INTERFACE I_HE_SolidAttenuatorAttentuationLengthDatabase EXTENDS I_Fallible


METHOD GetAttenuationLength
VAR_INPUT
    PhotonEnergy : I_QuantityLREAL;
    MaterialName : T_MaxString;
    AttenuationLengthOutput : I_QuantityLREALPublic;
END_VAR
END_METHOD

END_INTERFACE

(* stored: Version 1.1.0.1
   Itf I_HE_SolidAttenuatorAttentuationLengthDatabase: Id {06dfad59-b310-4aa0-bb9c-06b6bb0d52ba}
   Method GetAttenuationLength: Id {858654b7-988b-4231-baf6-21f5258c6a63} *)
